//{attribute 'qualified_only'}
VAR_GLOBAL
END_VAR

(* stored: Version 1.1.0.1, ProductVersion 3.1.4022.18
   GVL GVL_Devices: Id {3ef1adf5-ba18-48c2-a083-7ec1a9d4dd63} *)
